// TIA Portal V20 export
FUNCTION_BLOCK "LER_Axis64Pos_InterlockSummary"   // FB32866, LAD
// stored: Access Published, MemoryReserve 100, SetENOAutomatically false
   VAR_INPUT
      enableManualCmds : Bool;
      activeJobNumber : DInt;
      interlockSource { ExternalAccessible := 'False'; ExternalVisible := 'False'; ExternalWritable := 'False'} : "LER_typeAxisInterlockSource";
   END_VAR
   VAR_OUTPUT
      interlockcGeneral : Bool;
   END_VAR
   VAR_IN_OUT
      moduleInterface : "LBC_typeAxis64PosInterface";
      controlNode : "LBC_typeAxis64PosControlNode";
   END_VAR
   VAR
      statProcessValuesCommands { S7_SetPoint := 'True'} : "LBC_typeAxis64PosControlNodeCommands";
      statAnyInterlockAlive { S7_SetPoint := 'True'} : Bool;
   END_VAR
   VAR CONSTANT
      TRUE : Bool := TRUE;
      FALSE : Bool := FALSE;
   END_VAR
BEGIN

REGION Network 1: Command Capture (HMI / ControlNode arbitration)
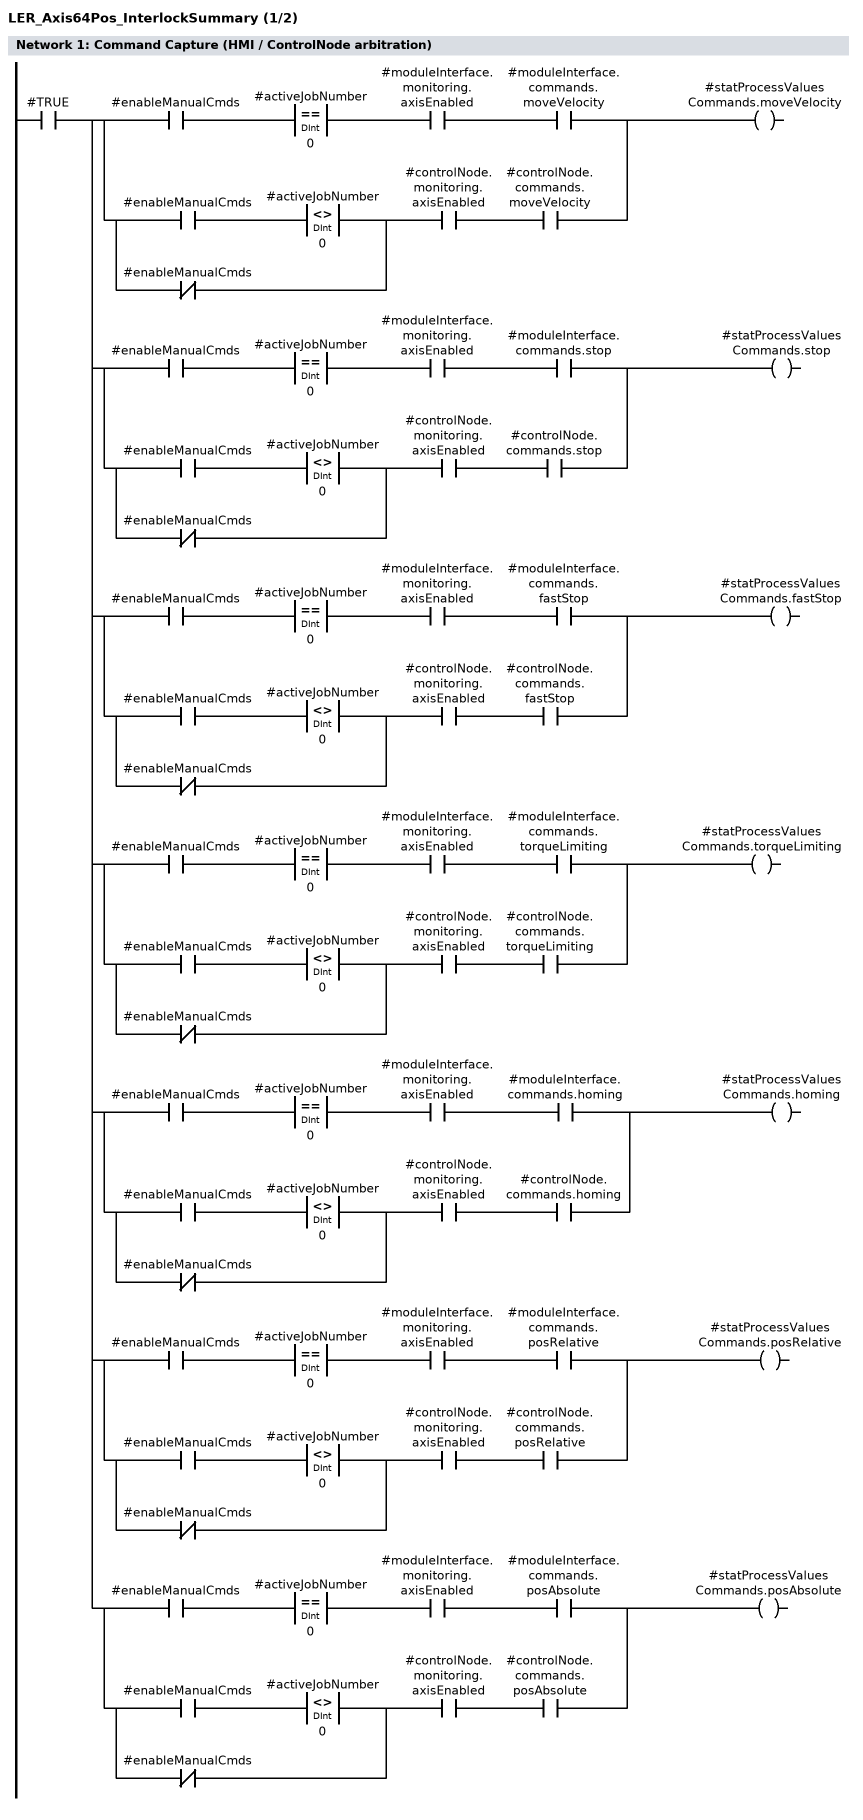
   RUNG wire#powerrail
      Contact( #TRUE )
      wire#w1
      Contact( #enableManualCmds )
      { S7_Templates := "SrcType := DInt" } EQ_Contact(in1 := #activeJobNumber, in2 := 0)
      Contact( #moduleInterface.monitoring.axisEnabled )
      Contact( #moduleInterface.commands.moveVelocity )
      wire#w2
      Coil( #statProcessValuesCommands.moveVelocity )
   END_RUNG
   RUNG wire#w1
      Contact( #enableManualCmds )
      { S7_Templates := "SrcType := DInt" } NE_Contact(in1 := #activeJobNumber, in2 := 0)
      wire#w3
      Contact( #controlNode.monitoring.axisEnabled )
      Contact( #controlNode.commands.moveVelocity )
   END_RUNG wire#w2
   RUNG wire#w1
      I_Contact( #enableManualCmds )
   END_RUNG wire#w3
   RUNG wire#w1
      Contact( #enableManualCmds )
      { S7_Templates := "SrcType := DInt" } EQ_Contact(in1 := #activeJobNumber, in2 := 0)
      Contact( #moduleInterface.monitoring.axisEnabled )
      Contact( #moduleInterface.commands.stop )
      wire#w4
      Coil( #statProcessValuesCommands.stop )
   END_RUNG
   RUNG wire#w1
      Contact( #enableManualCmds )
      { S7_Templates := "SrcType := DInt" } NE_Contact(in1 := #activeJobNumber, in2 := 0)
      wire#w5
      Contact( #controlNode.monitoring.axisEnabled )
      Contact( #controlNode.commands.stop )
   END_RUNG wire#w4
   RUNG wire#w1
      I_Contact( #enableManualCmds )
   END_RUNG wire#w5
   RUNG wire#w1
      Contact( #enableManualCmds )
      { S7_Templates := "SrcType := DInt" } EQ_Contact(in1 := #activeJobNumber, in2 := 0)
      Contact( #moduleInterface.monitoring.axisEnabled )
      Contact( #moduleInterface.commands.fastStop )
      wire#w6
      Coil( #statProcessValuesCommands.fastStop )
   END_RUNG
   RUNG wire#w1
      Contact( #enableManualCmds )
      { S7_Templates := "SrcType := DInt" } NE_Contact(in1 := #activeJobNumber, in2 := 0)
      wire#w7
      Contact( #controlNode.monitoring.axisEnabled )
      Contact( #controlNode.commands.fastStop )
   END_RUNG wire#w6
   RUNG wire#w1
      I_Contact( #enableManualCmds )
   END_RUNG wire#w7
   RUNG wire#w1
      Contact( #enableManualCmds )
      { S7_Templates := "SrcType := DInt" } EQ_Contact(in1 := #activeJobNumber, in2 := 0)
      Contact( #moduleInterface.monitoring.axisEnabled )
      Contact( #moduleInterface.commands.torqueLimiting )
      wire#w8
      Coil( #statProcessValuesCommands.torqueLimiting )
   END_RUNG
   RUNG wire#w1
      Contact( #enableManualCmds )
      { S7_Templates := "SrcType := DInt" } NE_Contact(in1 := #activeJobNumber, in2 := 0)
      wire#w9
      Contact( #controlNode.monitoring.axisEnabled )
      Contact( #controlNode.commands.torqueLimiting )
   END_RUNG wire#w8
   RUNG wire#w1
      I_Contact( #enableManualCmds )
   END_RUNG wire#w9
   RUNG wire#w1
      Contact( #enableManualCmds )
      { S7_Templates := "SrcType := DInt" } EQ_Contact(in1 := #activeJobNumber, in2 := 0)
      Contact( #moduleInterface.monitoring.axisEnabled )
      Contact( #moduleInterface.commands.homing )
      wire#w10
      Coil( #statProcessValuesCommands.homing )
   END_RUNG
   RUNG wire#w1
      Contact( #enableManualCmds )
      { S7_Templates := "SrcType := DInt" } NE_Contact(in1 := #activeJobNumber, in2 := 0)
      wire#w11
      Contact( #controlNode.monitoring.axisEnabled )
      Contact( #controlNode.commands.homing )
   END_RUNG wire#w10
   RUNG wire#w1
      I_Contact( #enableManualCmds )
   END_RUNG wire#w11
   RUNG wire#w1
      Contact( #enableManualCmds )
      { S7_Templates := "SrcType := DInt" } EQ_Contact(in1 := #activeJobNumber, in2 := 0)
      Contact( #moduleInterface.monitoring.axisEnabled )
      Contact( #moduleInterface.commands.posRelative )
      wire#w12
      Coil( #statProcessValuesCommands.posRelative )
   END_RUNG
   RUNG wire#w1
      Contact( #enableManualCmds )
      { S7_Templates := "SrcType := DInt" } NE_Contact(in1 := #activeJobNumber, in2 := 0)
      wire#w13
      Contact( #controlNode.monitoring.axisEnabled )
      Contact( #controlNode.commands.posRelative )
   END_RUNG wire#w12
   RUNG wire#w1
      I_Contact( #enableManualCmds )
   END_RUNG wire#w13
   RUNG wire#w1
      Contact( #enableManualCmds )
      { S7_Templates := "SrcType := DInt" } EQ_Contact(in1 := #activeJobNumber, in2 := 0)
      Contact( #moduleInterface.monitoring.axisEnabled )
      Contact( #moduleInterface.commands.posAbsolute )
      wire#w14
      Coil( #statProcessValuesCommands.posAbsolute )
   END_RUNG
   RUNG wire#w1
      Contact( #enableManualCmds )
      { S7_Templates := "SrcType := DInt" } NE_Contact(in1 := #activeJobNumber, in2 := 0)
      wire#w15
      Contact( #controlNode.monitoring.axisEnabled )
      Contact( #controlNode.commands.posAbsolute )
   END_RUNG wire#w14
   RUNG wire#w1
      I_Contact( #enableManualCmds )
   END_RUNG wire#w15
   // the same network as SCL:
   #statProcessValuesCommands.moveVelocity := #TRUE AND ((#enableManualCmds AND (#activeJobNumber = 0) AND #moduleInterface.monitoring.axisEnabled AND #moduleInterface.commands.moveVelocity) OR (((#enableManualCmds AND (#activeJobNumber <> 0)) OR NOT #enableManualCmds) AND #controlNode.monitoring.axisEnabled AND #controlNode.commands.moveVelocity));
   #statProcessValuesCommands.stop := #TRUE AND ((#enableManualCmds AND (#activeJobNumber = 0) AND #moduleInterface.monitoring.axisEnabled AND #moduleInterface.commands.stop) OR (((#enableManualCmds AND (#activeJobNumber <> 0)) OR NOT #enableManualCmds) AND #controlNode.monitoring.axisEnabled AND #controlNode.commands.stop));
   #statProcessValuesCommands.fastStop := #TRUE AND ((#enableManualCmds AND (#activeJobNumber = 0) AND #moduleInterface.monitoring.axisEnabled AND #moduleInterface.commands.fastStop) OR (((#enableManualCmds AND (#activeJobNumber <> 0)) OR NOT #enableManualCmds) AND #controlNode.monitoring.axisEnabled AND #controlNode.commands.fastStop));
   #statProcessValuesCommands.torqueLimiting := #TRUE AND ((#enableManualCmds AND (#activeJobNumber = 0) AND #moduleInterface.monitoring.axisEnabled AND #moduleInterface.commands.torqueLimiting) OR (((#enableManualCmds AND (#activeJobNumber <> 0)) OR NOT #enableManualCmds) AND #controlNode.monitoring.axisEnabled AND #controlNode.commands.torqueLimiting));
   #statProcessValuesCommands.homing := #TRUE AND ((#enableManualCmds AND (#activeJobNumber = 0) AND #moduleInterface.monitoring.axisEnabled AND #moduleInterface.commands.homing) OR (((#enableManualCmds AND (#activeJobNumber <> 0)) OR NOT #enableManualCmds) AND #controlNode.monitoring.axisEnabled AND #controlNode.commands.homing));
   #statProcessValuesCommands.posRelative := #TRUE AND ((#enableManualCmds AND (#activeJobNumber = 0) AND #moduleInterface.monitoring.axisEnabled AND #moduleInterface.commands.posRelative) OR (((#enableManualCmds AND (#activeJobNumber <> 0)) OR NOT #enableManualCmds) AND #controlNode.monitoring.axisEnabled AND #controlNode.commands.posRelative));
   #statProcessValuesCommands.posAbsolute := #TRUE AND ((#enableManualCmds AND (#activeJobNumber = 0) AND #moduleInterface.monitoring.axisEnabled AND #moduleInterface.commands.posAbsolute) OR (((#enableManualCmds AND (#activeJobNumber <> 0)) OR NOT #enableManualCmds) AND #controlNode.monitoring.axisEnabled AND #controlNode.commands.posAbsolute));
END_REGION

REGION Network 2: Command Parameter Transfer
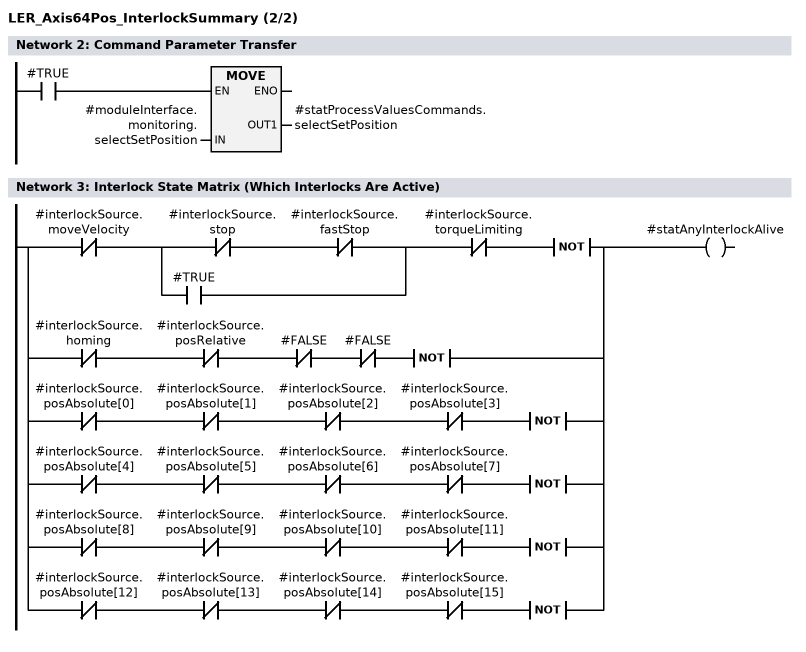
   RUNG wire#powerrail
      Contact( #TRUE )
      Move(in := #moduleInterface.monitoring.selectSetPosition, out1 => #statProcessValuesCommands.selectSetPosition)
   END_RUNG
   // the same network as SCL:
   IF #TRUE THEN
       #statProcessValuesCommands.selectSetPosition := #moduleInterface.monitoring.selectSetPosition;
   END_IF;
END_REGION

REGION Network 3: Interlock State Matrix (Which Interlocks Are Active)
   RUNG wire#powerrail
      I_Contact( #interlockSource.moveVelocity )
      wire#w1
      I_Contact( #interlockSource.stop )
      I_Contact( #interlockSource.fastStop )
      wire#w2
      I_Contact( #interlockSource.torqueLimiting )
      Not()
      wire#w3
      Coil( #statAnyInterlockAlive )
   END_RUNG
   RUNG wire#w1
      Contact( #TRUE )
   END_RUNG wire#w2
   RUNG wire#powerrail
      I_Contact( #interlockSource.homing )
      I_Contact( #interlockSource.posRelative )
      I_Contact( #FALSE )
      I_Contact( #FALSE )
      Not()
   END_RUNG wire#w3
   RUNG wire#powerrail
      I_Contact( #interlockSource.posAbsolute[0] )
      I_Contact( #interlockSource.posAbsolute[1] )
      I_Contact( #interlockSource.posAbsolute[2] )
      I_Contact( #interlockSource.posAbsolute[3] )
      Not()
   END_RUNG wire#w3
   RUNG wire#powerrail
      I_Contact( #interlockSource.posAbsolute[4] )
      I_Contact( #interlockSource.posAbsolute[5] )
      I_Contact( #interlockSource.posAbsolute[6] )
      I_Contact( #interlockSource.posAbsolute[7] )
      Not()
   END_RUNG wire#w3
   RUNG wire#powerrail
      I_Contact( #interlockSource.posAbsolute[8] )
      I_Contact( #interlockSource.posAbsolute[9] )
      I_Contact( #interlockSource.posAbsolute[10] )
      I_Contact( #interlockSource.posAbsolute[11] )
      Not()
   END_RUNG wire#w3
   RUNG wire#powerrail
      I_Contact( #interlockSource.posAbsolute[12] )
      I_Contact( #interlockSource.posAbsolute[13] )
      I_Contact( #interlockSource.posAbsolute[14] )
      I_Contact( #interlockSource.posAbsolute[15] )
      Not()
   END_RUNG wire#w3
   // the same network as SCL:
   #statAnyInterlockAlive := NOT (NOT #interlockSource.moveVelocity AND ((NOT #interlockSource.stop AND NOT #interlockSource.fastStop) OR #TRUE) AND NOT #interlockSource.torqueLimiting) OR NOT (NOT #interlockSource.homing AND NOT #interlockSource.posRelative AND NOT #FALSE AND NOT #FALSE) OR NOT (NOT #interlockSource.posAbsolute[0] AND NOT #interlockSource.posAbsolute[1] AND NOT #interlockSource.posAbsolute[2] AND NOT #interlockSource.posAbsolute[3]) OR NOT (NOT #interlockSource.posAbsolute[4] AND NOT #interlockSource.posAbsolute[5] AND NOT #interlockSource.posAbsolute[6] AND NOT #interlockSource.posAbsolute[7]) OR NOT (NOT #interlockSource.posAbsolute[8] AND NOT #interlockSource.posAbsolute[9] AND NOT #interlockSource.posAbsolute[10] AND NOT #interlockSource.posAbsolute[11]) OR NOT (NOT #interlockSource.posAbsolute[12] AND NOT #interlockSource.posAbsolute[13] AND NOT #interlockSource.posAbsolute[14] AND NOT #interlockSource.posAbsolute[15]);
END_REGION

REGION Network 4 (SCL): Active Motion Interlock Arbitration
   IF #statProcessValuesCommands.moveVelocity OR (#controlNode.monitoring.moveVelocitySelected AND #controlNode.monitoring.commandBusy) THEN
       #interlockcGeneral := #interlockSource.moveVelocity;

   // ELSIF #statProcessValuesCommands.stop AND (#controlNode.monitoring.stopSelected AND #controlNode.monitoring.commandDone) THEN
   //     #interlockcGeneral := #interlockSource.stop;

   // ELSIF #statProcessValuesCommands.fastStop AND (#controlNode.monitoring.fastStopSelected AND #controlNode.monitoring.commandDone) THEN
   //     #interlockcGeneral := #interlockSource.fastStop;

   ELSIF #statProcessValuesCommands.torqueLimiting OR (#controlNode.monitoring.torqueLimitingSelected AND #controlNode.monitoring.commandBusy) THEN
       #interlockcGeneral := #interlockSource.torqueLimiting;

   ELSIF #statProcessValuesCommands.homing OR (#controlNode.monitoring.homingSelected AND #controlNode.monitoring.commandBusy) THEN
       #interlockcGeneral := #interlockSource.homing;

   ELSIF #statProcessValuesCommands.posRelative OR (#controlNode.monitoring.posRelativeSelected AND #controlNode.monitoring.commandBusy) THEN
       #interlockcGeneral := #interlockSource.posRelative;

   ELSIF #statProcessValuesCommands.posAbsolute OR (#controlNode.monitoring.posAbsoluteSelected AND #controlNode.monitoring.commandBusy) THEN

       CASE #statProcessValuesCommands.selectSetPosition OF
           0:
               #interlockcGeneral := #interlockSource.posAbsolute[0];
           1:
               #interlockcGeneral := #interlockSource.posAbsolute[1];
           2:
               #interlockcGeneral := #interlockSource.posAbsolute[2];
           3:
               #interlockcGeneral := #interlockSource.posAbsolute[3];
           4:
               #interlockcGeneral := #interlockSource.posAbsolute[4];
           5:
               #interlockcGeneral := #interlockSource.posAbsolute[5];
           6:
               #interlockcGeneral := #interlockSource.posAbsolute[6];
           7:
               #interlockcGeneral := #interlockSource.posAbsolute[7];
           8:
               #interlockcGeneral := #interlockSource.posAbsolute[8];
           9:
               #interlockcGeneral := #interlockSource.posAbsolute[9];
           10:
               #interlockcGeneral := #interlockSource.posAbsolute[10];
           11:
               #interlockcGeneral := #interlockSource.posAbsolute[11];
           12:
               #interlockcGeneral := #interlockSource.posAbsolute[12];
           13:
               #interlockcGeneral := #interlockSource.posAbsolute[13];
           14:
               #interlockcGeneral := #interlockSource.posAbsolute[14];
           15:
               #interlockcGeneral := #interlockSource.posAbsolute[15];

       END_CASE;

   ELSE
       #interlockcGeneral := #statAnyInterlockAlive;
   END_IF;
END_REGION
END_FUNCTION_BLOCK
